{attribute 'GeneratedUsingTerminal: EL2595-0000-0019'}
{attribute addProperty BoxType "EL2595-0000-0019"}
{attribute addProperty Description "EL2595 1Ch. LED constant current terminal"}
{attribute addProperty Physics "KK"}
{attribute addProperty Id "DOX_StatusAT %I*DOX_Status_F52B34D37DOX_ControlAT %Q*DOX_Control_75D5C9E23WcStateAT %I*WcState_9091E0EB2InfoDataAT %I*InfoData_32EB74EA10"}
{attribute addProperty CRC "1425051988"}
{attribute addProperty Size "22"}
TYPE EL2595_54F09154 EXTENDS EtcSlaveTerminalBase_947E5A46 :
STRUCT
	{attribute addProperty Name "DOX_Status"}
	DOX_Status : DOX_Status_F52B34D3;
	{attribute addProperty Name "DOX_Control"}
	DOX_Control : DOX_Control_75D5C9E2;
	{attribute addProperty Name "WcState"}
	WcState : WcState_9091E0EB;
	{attribute addProperty Name "InfoData"}
	InfoData : InfoData_32EB74EA;
END_STRUCT
END_TYPE

(* stored: Version 1.2.0.0, ProductVersion 3.1.4024.9
   DUT EL2595_54F09154: Id {3d324843-4353-4334-bec7-173ed3caa447} *)
